TYPE Range :
STRUCT
	Bottom : LREAL;
	Top : LREAL;
END_STRUCT
END_TYPE

(* stored: Version 1.1.0.1
   DUT Range: Id {a9b63f91-5b34-0f99-353a-641d18d0a4b5} *)
